TYPE ST_SettingsServo :
STRUCT
	fHomeOffset : LREAL := 0.0; //[mm]
	fPositionBias : LREAL := 0.0; //[mm]
	
	fStopDec : LREAL := 10.0; //[mm/s^2]
	fStopJrk : LREAL := 100.0; //[mm/s^3]
	
	fJogVel : LREAL := 1.0; //[mm/s]
	fJogAcc : LREAL := 10.0; //[mm/s^2]
	fJogDec : LREAL := 10.0; //[mm/s^2]
	fJogJrk : LREAL := 100.0; //[mm/s^3]
	
	fAbsPosPos : LREAL := 0.0; //[mm]
	fAbsPosVel : LREAL := 1.0; //[mm/s]
	fAbsPosAcc : LREAL := 10.0; //[mm/s^2]
	fAbsPosDec : LREAL := 10.0; //[mm/s^2]
	fAbsPosJrk : LREAL := 100.0; //[mm/s^3]
END_STRUCT
END_TYPE

(* stored: Version 1.1.0.1, ProductVersion 3.1.4024.12
   DUT ST_SettingsServo: Id {ed6a1034-fbc2-4d8e-a32e-f51a7b4f2923} *)
